INTERFACE I_AO_percentage

PROPERTY max_value : real
GET
END_GET
SET
END_SET
END_PROPERTY

PROPERTY min_value : real
GET
END_GET
SET
END_SET
END_PROPERTY

PROPERTY value : real
GET
END_GET
END_PROPERTY

END_INTERFACE

(* stored: Version 1.1.0.1, ProductVersion 3.1.4024.6
   Itf I_AO_percentage: Id {f94ffe78-2e7a-0d2f-0a72-8efbd9ab635a}
   Property max_value: Id {725099ed-c625-06bb-193c-a5d0e309af5f}
   Get Get: Id {c821549b-7648-01b5-0cad-64b1a6da1f43}
   Set Set: Id {3cef5204-257f-0101-3fde-7a5f06a9dfae}
   Property min_value: Id {7ae42cf2-5942-04cc-207d-5b9f53dcd8bf}
   Get Get: Id {9e03194b-fdae-03e4-1873-b624ea1e58c1}
   Set Set: Id {abfd66c0-0957-0a54-2ee3-ce4f5b2eab0a}
   Property value: Id {b978c758-cec7-0c15-17a1-f9f1649c5f0a}
   Get Get: Id {68d58029-6dd8-013b-1e1c-69aa7c8f8189} *)
